Omron CX-Programmer project NewProject (CX-Programmer 9.03)

# PLC NewPLC1: CP1L L

## Global symbols (name address type ; comment)
1.01 BOOL  ; Contoh NOR
1.00 BOOL  ; Contoh NAND
0.00 BOOL  ; 1
0.01 BOOL  ; 2
0.02 BOOL  ; 3
0.03 BOOL  ; 4

## Program NewProgram1 (cyclic task 0)

### Section Section1

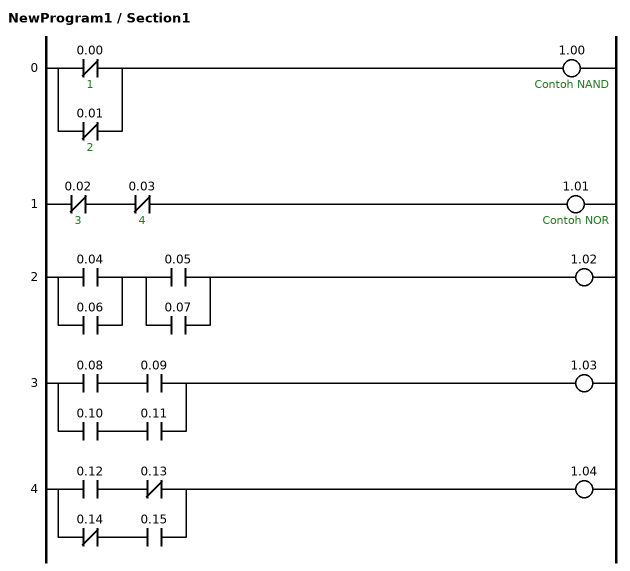
; rung 0
LDNOT 0.00  ; 1
ORNOT 0.01  ; 2
OUT 1.00  ; Contoh NAND
; rung 1
LDNOT 0.02  ; 3
ANDNOT 0.03  ; 4
OUT 1.01  ; Contoh NOR
; rung 2
LD 0.04
OR 0.06
LD 0.05
OR 0.07
ANDLD
OUT 1.02
; rung 3
LD 0.08
AND 0.09
LD 0.10
AND 0.11
ORLD
OUT 1.03
; rung 4
LD 0.12
ANDNOT 0.13
LDNOT 0.14
AND 0.15
ORLD
OUT 1.04

### Section END
; rung 0
END(001)